Staubli VAL3: exeMove_pulseDO.pgx

program exeMove_pulseDO(num x_nAdvMoveIndex, num x_nMoveId, point x_pPoint, tool x_tTool, num x_nDistance, num x_nPulseLength, dio x_dDio)
  local num l_givenId
  local num l_nDistance
  local num l_nMoveId
begin

  //I want to see the tool entering the zone
  //so at first I must be out
  wait(distance(position(here(x_tTool,world),world),position(x_pPoint,world))>=x_nDistance or roundDown(getMoveId())>roundDown(x_nMoveId))
  //then I go inside
  wait((distance(position(here(x_tTool,world),world),position(x_pPoint,world))<x_nDistance and roundDown(getMoveId())==roundDown(x_nMoveId)) or roundDown(getMoveId())>roundDown(x_nMoveId))

  if distance(position(here(x_tTool,world),world),position(x_pPoint,world))<x_nDistance
    //logMsg("libSignals/exeMove_PulseDO->success")
    call pulse(x_dDio,x_nPulseLength)
  elseIf roundDown(getMoveId())>roundDown(x_nMoveId)
    //the tool never passed close enough to x_pPoint
    logMsg("libSignals/exeMove_PulseDO->fail")
  endIf

  call freeAdvMove(x_nAdvMoveIndex)

end
